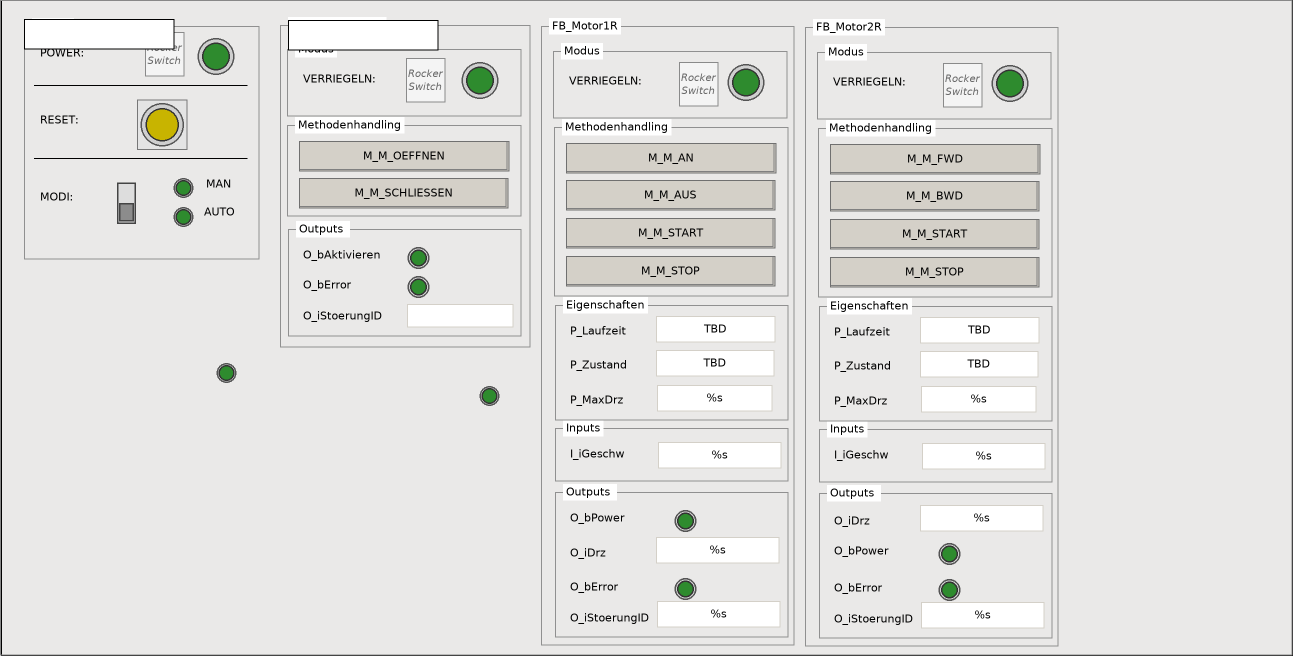
VISUALIZATION Aktoren  // 1293x656
    Rectangle (1,0 1292x656)
    GroupBox (280,17 250x330), "FB_Magnetventil"
        Textfield (127,287 106x23), text variable: Reaktoranlage.VENTIL.O_iStoerungID
    GroupBox (287,41 234x75), "Modus"
        Label (13,23 150x30), "VERRIEGELN:"
        Lamp1 (172,18 42x43), variable: Reaktoranlage.VENTIL.I_bVerriegeln, style: Lamp-Lamp1-Green
        Lamp1 (191,340 23x30), style: Lamp-Lamp1-Green
    RockerSwitch (406,58 39x44), variable: Reaktoranlage.VENTIL.I_bVerriegeln, behaviour: TOGGLE, style: Switch-RockerSwitch-Gray
    GroupBox (287,117 234x99), "Methodenhandling"
        Rectangle (-530,-100 150x30)
        Button (12,24 210x30), "M_M_OEFFNEN"
            OnMouseClick: execute { Reaktoranlage.VENTIL.M_M_OEFFNEN(); }
        Button (12,61 209x30), "M_M_SCHLIESSEN"
            OnMouseClick: execute { Reaktoranlage.VENTIL.M_M_SCHLIESSEN(); }
    GroupBox (288,221 233x115), "Outputs"
        Label (12,19 150x30), "O_bAktivieren"
        Label (12,49 150x30), "O_bError"
        Label (12,80 150x30), "O_iStoerungID"
        Lamp1 (118,22 25x30), variable: Reaktoranlage.VENTIL.O_bAktivieren, style: Lamp-Lamp1-Green
        Lamp1 (118,51 25x30), variable: Reaktoranlage.VENTIL.O_bError, style: Lamp-Lamp1-Green
    GroupBox (24,18 235x241), "Modus"
        Label (13,20 150x30), "POWER:"
        RockerSwitch (121,14 39x44), variable: Reaktoranlage.Modus.I_bPower, behaviour: TOGGLE, style: Switch-RockerSwitch-Gray
        Label (13,164 150x30), "MODI:"
        DipSwitch (82,161 41x48), variable: Reaktoranlage.Modus.I_bMode, behaviour: TOGGLE, style: Switch-DipSwitch-Gray
        Lamp1 (148,155 23x30), variable: Reaktoranlage.Modus.O_bMAN, style: Lamp-Lamp1-Green
        Lamp1 (148,184 23x30), variable: Reaktoranlage.Modus.O_bAUTO, style: Lamp-Lamp1-Green
        Label (177,179 46x30), "AUTO"
        Lamp1 (191,340 23x30), style: Lamp-Lamp1-Green
        Line (10,67) (223,67)
        Lamp1 (171,17 42x43), variable: Reaktoranlage.Modus.I_bPower, style: Lamp-Lamp1-Green
        Label (179,151 46x30), "MAN"
        Label (13,87 150x30), "RESET:"
        PushSwitch (113,80 50x53), variable: GVL.VIS_SysReset, behaviour: TAP, style: Switch-PushSwitch-Yellow
        Line (10,140) (223,140)
    GroupBox (541,18 253x627), "FB_Motor1R"
        GroupBox (12,25 234x75), "Modus"
            Label (13,23 150x30), "VERRIEGELN:"
            Lamp1 (172,18 42x43), variable: Reaktoranlage.RUEHRER.I_bVerriegeln, style: Lamp-Lamp1-Green
            Lamp1 (191,340 23x30), style: Lamp-Lamp1-Green
            RockerSwitch (126,19 39x44), variable: Reaktoranlage.RUEHRER.I_bVerriegeln, behaviour: TOGGLE, style: Switch-RockerSwitch-Gray
        GroupBox (13,101 234x177), "Methodenhandling"
            Rectangle (-530,-100 150x30)
            Button (12,24 210x30), "M_M_AN"
                OnMouseClick: execute { Reaktoranlage.RUEHRER.M_M_AN(); }
            Button (12,61 209x30), "M_M_AUS"
                OnMouseClick: execute { Reaktoranlage.RUEHRER.M_M_AUS(); }
            Button (12,99 209x30), "M_M_START"
                OnMouseClick: execute { Reaktoranlage.RUEHRER.M_M_START(); }
            Button (12,137 209x30), "M_M_STOP"
                OnMouseClick: execute { Reaktoranlage.RUEHRER.M_M_STOP(); }
        GroupBox (14,402 233x61), "Inputs"
            Label (12,19 150x30), "I_iGeschw"
            Textfield (103,22 123x26), "%s", text variable: Reaktoranlage.RUEHRER.I_iGeschw
                OnMouseClick: write Reaktoranlage.RUEHRER.I_iGeschw via Edit, min 0
        GroupBox (14,279 233x123), "Eigenschaften"
            Label (12,19 150x30), "P_Laufzeit"
            Label (12,88 150x30), "P_MaxDrz"
            Label (12,53 150x30), "P_Zustand"
            Textfield (101,53 118x26), "TBD", input disabled if: TRUE
            Textfield (102,88 115x26), "%s", text variable: Reaktoranlage.RUEHRER.V_DrzMax
                OnMouseClick: execute { Reaktoranlage.RUEHRER.P_MaxDrz := 100; }
            Textfield (101,19 119x26), "TBD", input disabled if: TRUE
        GroupBox (14,466 233x153), "Outputs"
            Label (12,19 150x30), "O_bPower"
            Label (12,88 150x30), "O_bError"
            Label (12,119 150x30), "O_iStoerungID"
            Lamp1 (118,22 25x30), variable: Reaktoranlage.RUEHRER.O_bPower, style: Lamp-Lamp1-Green
            Lamp1 (118,90 25x30), variable: Reaktoranlage.RUEHRER.O_bError, style: Lamp-Lamp1-Green
            Textfield (101,53 123x26), "%s", text variable: Reaktoranlage.RUEHRER.O_iDrz, input disabled if: TRUE
            Textfield (102,117 123x26), "%s", text variable: Reaktoranlage.RUEHRER.O_iStoerungID, input disabled if: TRUE
            Label (12,54 150x30), "O_iDrz"
    GroupBox (805,19 253x627), "FB_Motor2R"
        GroupBox (12,25 234x75), "Modus"
            Label (13,23 150x30), "VERRIEGELN:"
            Lamp1 (172,18 42x43), variable: Reaktoranlage.RUEHRER.I_bVerriegeln, style: Lamp-Lamp1-Green
            Lamp1 (191,340 23x30), style: Lamp-Lamp1-Green
            RockerSwitch (126,19 39x44), variable: Reaktoranlage.RUEHRER.I_bVerriegeln, behaviour: TOGGLE, style: Switch-RockerSwitch-Gray
        GroupBox (13,101 234x177), "Methodenhandling"
            Rectangle (-530,-100 150x30)
            Button (12,24 210x30), "M_M_FWD"
            Button (12,61 209x30), "M_M_BWD"
            Button (12,99 209x30), "M_M_START"
            Button (12,137 209x30), "M_M_STOP"
        GroupBox (14,402 233x61), "Inputs"
            Label (12,19 150x30), "I_iGeschw"
            Textfield (103,22 123x26), "%s", text variable: Reaktoranlage.RUEHRER.I_iGeschw
                OnMouseClick: write Reaktoranlage.RUEHRER.I_iGeschw via Edit, min 0
        GroupBox (14,279 233x123), "Eigenschaften"
            Label (12,19 150x30), "P_Laufzeit"
            Label (12,88 150x30), "P_MaxDrz"
            Label (12,53 150x30), "P_Zustand"
            Textfield (101,53 118x26), "TBD", input disabled if: TRUE
            Textfield (102,88 115x26), "%s", text variable: Reaktoranlage.RUEHRER.V_DrzMax
                OnMouseClick: execute { Reaktoranlage.PUMPE.P_MaxDrz := 100; }
            Textfield (101,19 119x26), "TBD", input disabled if: TRUE
        GroupBox (14,466 233x153), "Outputs"
            Label (12,51 150x30), "O_bPower"
            Label (12,88 150x30), "O_bError"
            Label (12,119 150x30), "O_iStoerungID"
            Lamp1 (118,54 25x30), variable: Reaktoranlage.RUEHRER.O_bPower, style: Lamp-Lamp1-Green
            Lamp1 (118,90 25x30), variable: Reaktoranlage.RUEHRER.O_bError, style: Lamp-Lamp1-Green
            Textfield (101,20 123x26), "%s", text variable: Reaktoranlage.RUEHRER.O_iDrz, input disabled if: TRUE
            Textfield (102,117 123x26), "%s", text variable: Reaktoranlage.RUEHRER.O_iStoerungID, input disabled if: TRUE
            Label (12,21 150x30), "O_iDrz"
END_VISUALIZATION

(* stored: Version 1.1.0.1, ProductVersion 3.1.4024.12
   Visu Aktoren: Id {ac277a63-1cee-4a87-a068-9fd3f4af00ac} *)
